// TIA Portal V17 export
// export: Created 2026-04-13T11:12:44.2249496Z, ExportSetting WithDefaults, DisplayName Totally Integrated Automation Portal, DisplayVersion V17 Update 4, DisplayName TIA Portal Openness, DisplayVersion V17 Update 4, DisplayName TIA Portal Version Control Interface, DisplayVersion V17, DisplayName SINAMICS Startdrive Advanced, DisplayVersion V17, DisplayName SINAMICS Startdrive G130, G150, S120, S150, SINAMICS MV, S210, DisplayVersion V17, DisplayName SINAMICS Startdrive G110M, G120, G120C, G120D, G120P, G115D, DisplayVersion V17, DisplayName STEP 7 Professional, DisplayVersion V17 Update 4, DisplayName STEP 7 Safety, DisplayVersion V17, DisplayName WinCC Professional, DisplayVersion V17 Update 4
FUNCTION_BLOCK "16-普通脉冲"   // FB53, SCL
{ S7_Optimized_Access := 'TRUE' }
VERSION : 0.1
// stored: AutoNumber true, IsIECCheckEnabled false, IsRetainMemResEnabled false, MemoryReserve 100, SetENOAutomatically false, UDAEnableTagReadback false
   VAR_INPUT
      模式设定 : Real;
      QD : Bool;
      On_Time : Real;
      Stop_Time : Real;
      Num : Int;
   END_VAR
   VAR_OUTPUT
      Output_1 : Bool;
      Output_2 : Bool;
      Output_3 : Bool;
      Output_4 : Bool;
      Output_5 : Bool;
      Output_6 : Bool;
      Output_7 : Bool;
      Output_8 : Bool;
      Num_now : Int;
   END_VAR
   VAR
      Stoptime : Time;
      WorkTime : Time;
      TON_ON : Array[1..10] of TON_TIME;
      TON_OFF : Array[1..10] of TON_TIME;
   END_VAR
BEGIN

   IF #模式设定 = 1.0  OR #模式设定 = 2.0  THEN
       #Stoptime := DINT_TO_TIME(REAL_TO_DINT(#Stop_Time * 1000.0));
       //#WorkTime := DINT_TO_TIME(REAL_TO_DINT(#On_Time * 1000));
        #WorkTime := REAL_TO_DINT(#On_Time);

       IF NOT #QD THEN
           #Num_now := 0;
       ELSE

           IF #Num <= 12 THEN
               #Num_now := #Num;
           ELSE
               #Num_now := 12;
           END_IF;

       END_IF;



       CASE #Num_now OF
           1:
               #TON_ON[1](IN := #QD AND NOT #TON_OFF[1].Q,
                          PT := #WorkTime);
               #TON_OFF[1](IN := #QD AND #TON_ON[1].Q,
                           PT := #Stoptime);


               #Output_1 := #QD AND NOT #TON_ON[1].Q;


           2:  // Statement section case 1
               #TON_ON[1](IN := #QD AND NOT #TON_OFF[2].Q,
                          PT := #WorkTime);
               #TON_OFF[1](IN := #QD AND #TON_ON[1].Q,
                           PT := #Stoptime);
               #TON_ON[2](IN := #QD AND #TON_ON[1].Q AND #TON_OFF[1].Q,
                          PT := #WorkTime);
               #TON_OFF[2](IN := #QD AND #TON_ON[1].Q AND #TON_OFF[1].Q AND #TON_ON[2].Q,
                           PT := #Stoptime);

               #Output_1 := #QD AND NOT #TON_ON[1].Q;
               #Output_2 := #QD AND #TON_ON[1].Q AND #TON_OFF[1].Q AND NOT #TON_ON[2].Q;

           3:  // Statement section case 2 to 4
               #TON_ON[1](IN := #QD AND NOT #TON_OFF[3].Q,
                          PT := #WorkTime);
               #TON_OFF[1](IN := #QD AND #TON_ON[1].Q,
                           PT := #Stoptime);
               #TON_ON[2](IN := #QD AND #TON_ON[1].Q AND #TON_OFF[1].Q,
                          PT := #WorkTime);
               #TON_OFF[2](IN := #QD AND #TON_ON[1].Q AND #TON_OFF[1].Q AND #TON_ON[2].Q,
                           PT := #Stoptime);
               #TON_ON[3](IN := #QD AND #TON_ON[1].Q AND #TON_OFF[1].Q AND #TON_ON[2].Q AND #TON_OFF[2].Q,
                          PT := #WorkTime);
               #TON_OFF[3](IN := #QD AND #TON_ON[1].Q AND #TON_OFF[1].Q AND #TON_ON[2].Q AND #TON_OFF[2].Q AND #TON_ON[3].Q,
                           PT := #Stoptime);
               #Output_1 := #QD AND NOT #TON_ON[1].Q;
               #Output_2 := #QD AND #TON_ON[1].Q AND #TON_OFF[1].Q AND NOT #TON_ON[2].Q;
               #Output_3 := #QD AND #TON_ON[1].Q AND #TON_OFF[1].Q AND #TON_ON[2].Q AND #TON_OFF[2].Q AND NOT #TON_ON[3].Q;
           4:  // Statement section case 2 to 4
               #TON_ON[1](IN := #QD AND NOT #TON_OFF[4].Q,
                          PT := #WorkTime);
               #TON_OFF[1](IN := #QD AND #TON_ON[1].Q,
                           PT := #Stoptime);
               #TON_ON[2](IN := #QD AND #TON_ON[1].Q AND #TON_OFF[1].Q,
                          PT := #WorkTime);
               #TON_OFF[2](IN := #QD AND #TON_ON[1].Q AND #TON_OFF[1].Q AND #TON_ON[2].Q,
                           PT := #Stoptime);
               #TON_ON[3](IN := #QD AND #TON_ON[1].Q AND #TON_OFF[1].Q AND #TON_ON[2].Q AND #TON_OFF[2].Q,
                          PT := #WorkTime);
               #TON_OFF[3](IN := #QD AND #TON_ON[1].Q AND #TON_OFF[1].Q AND #TON_ON[2].Q AND #TON_OFF[2].Q AND #TON_ON[3].Q,
                           PT := #Stoptime);

               #TON_ON[4](IN := #QD AND #TON_ON[1].Q AND #TON_OFF[1].Q AND #TON_ON[2].Q AND #TON_OFF[2].Q AND #TON_ON[3].Q AND #TON_OFF[3].Q,
                          PT := #WorkTime);
               #TON_OFF[4](IN := #QD AND #TON_ON[1].Q AND #TON_OFF[1].Q AND #TON_ON[2].Q AND #TON_OFF[2].Q AND #TON_ON[3].Q AND #TON_OFF[3].Q AND #TON_ON[4].Q,
                           PT := #Stoptime);


               #Output_1 := #QD AND NOT #TON_ON[1].Q;
               #Output_2 := #QD AND #TON_ON[1].Q AND #TON_OFF[1].Q AND NOT #TON_ON[2].Q;
               #Output_3 := #QD AND #TON_ON[1].Q AND #TON_OFF[1].Q AND #TON_ON[2].Q AND #TON_OFF[2].Q AND NOT #TON_ON[3].Q;
               #Output_4 := #QD AND #TON_ON[1].Q AND #TON_OFF[1].Q AND #TON_ON[2].Q AND #TON_OFF[2].Q AND #TON_ON[3].Q AND #TON_OFF[3].Q AND NOT #TON_ON[4].Q;

           5:  // Statement section case 2 to 4
               #TON_ON[1](IN := #QD AND NOT #TON_OFF[5].Q,
                          PT := #WorkTime);
               #TON_OFF[1](IN := #QD AND #TON_ON[1].Q,
                           PT := #Stoptime);
               #TON_ON[2](IN := #QD AND #TON_ON[1].Q AND #TON_OFF[1].Q,
                          PT := #WorkTime);
               #TON_OFF[2](IN := #QD AND #TON_ON[1].Q AND #TON_OFF[1].Q AND #TON_ON[2].Q,
                           PT := #Stoptime);
               #TON_ON[3](IN := #QD AND #TON_ON[1].Q AND #TON_OFF[1].Q AND #TON_ON[2].Q AND #TON_OFF[2].Q,
                          PT := #WorkTime);
               #TON_OFF[3](IN := #QD AND #TON_ON[1].Q AND #TON_OFF[1].Q AND #TON_ON[2].Q AND #TON_OFF[2].Q AND #TON_ON[3].Q,
                           PT := #Stoptime);

               #TON_ON[4](IN := #QD AND #TON_ON[1].Q AND #TON_OFF[1].Q AND #TON_ON[2].Q AND #TON_OFF[2].Q AND #TON_ON[3].Q AND #TON_OFF[3].Q,
                          PT := #WorkTime);
               #TON_OFF[4](IN := #QD AND #TON_ON[1].Q AND #TON_OFF[1].Q AND #TON_ON[2].Q AND #TON_OFF[2].Q AND #TON_ON[3].Q AND #TON_OFF[3].Q AND #TON_ON[4].Q,
                           PT := #Stoptime);

               #TON_ON[5](IN := #QD AND #TON_ON[1].Q AND #TON_OFF[1].Q AND #TON_ON[2].Q AND #TON_OFF[2].Q AND #TON_ON[3].Q AND #TON_OFF[3].Q AND #TON_ON[4].Q AND #TON_OFF[4].Q,
                          PT := #WorkTime);
               #TON_OFF[5](IN := #QD AND #TON_ON[1].Q AND #TON_OFF[1].Q AND #TON_ON[2].Q AND #TON_OFF[2].Q AND #TON_ON[3].Q AND #TON_OFF[3].Q AND #TON_ON[4].Q AND #TON_OFF[4].Q AND #TON_ON[5].Q,
                           PT := #Stoptime);


               #Output_1 := #QD AND NOT #TON_ON[1].Q;
               #Output_2 := #QD AND #TON_ON[1].Q AND #TON_OFF[1].Q AND NOT #TON_ON[2].Q;
               #Output_3 := #QD AND #TON_ON[1].Q AND #TON_OFF[1].Q AND #TON_ON[2].Q AND #TON_OFF[2].Q AND NOT #TON_ON[3].Q;
               #Output_4 := #QD AND #TON_ON[1].Q AND #TON_OFF[1].Q AND #TON_ON[2].Q AND #TON_OFF[2].Q AND #TON_ON[3].Q AND #TON_OFF[3].Q AND NOT #TON_ON[4].Q;
               #Output_5 := #QD AND #TON_ON[1].Q AND #TON_OFF[1].Q AND #TON_ON[2].Q AND #TON_OFF[2].Q AND #TON_ON[3].Q AND #TON_OFF[3].Q AND #TON_ON[4].Q AND #TON_OFF[4].Q AND NOT #TON_ON[5].Q;

           6:  // Statement section case 2 to 4
               #TON_ON[1](IN := #QD AND NOT #TON_OFF[6].Q,
                          PT := #WorkTime);
               #TON_OFF[1](IN := #QD AND #TON_ON[1].Q,
                           PT := #Stoptime);
               #TON_ON[2](IN := #QD AND #TON_ON[1].Q AND #TON_OFF[1].Q,
                          PT := #WorkTime);
               #TON_OFF[2](IN := #QD AND #TON_ON[1].Q AND #TON_OFF[1].Q AND #TON_ON[2].Q,
                           PT := #Stoptime);
               #TON_ON[3](IN := #QD AND #TON_ON[1].Q AND #TON_OFF[1].Q AND #TON_ON[2].Q AND #TON_OFF[2].Q,
                          PT := #WorkTime);
               #TON_OFF[3](IN := #QD AND #TON_ON[1].Q AND #TON_OFF[1].Q AND #TON_ON[2].Q AND #TON_OFF[2].Q AND #TON_ON[3].Q,
                           PT := #Stoptime);

               #TON_ON[4](IN := #QD AND #TON_ON[1].Q AND #TON_OFF[1].Q AND #TON_ON[2].Q AND #TON_OFF[2].Q AND #TON_ON[3].Q AND #TON_OFF[3].Q,
                          PT := #WorkTime);
               #TON_OFF[4](IN := #QD AND #TON_ON[1].Q AND #TON_OFF[1].Q AND #TON_ON[2].Q AND #TON_OFF[2].Q AND #TON_ON[3].Q AND #TON_OFF[3].Q AND #TON_ON[4].Q,
                           PT := #Stoptime);

               #TON_ON[5](IN := #QD AND #TON_ON[1].Q AND #TON_OFF[1].Q AND #TON_ON[2].Q AND #TON_OFF[2].Q AND #TON_ON[3].Q AND #TON_OFF[3].Q AND #TON_ON[4].Q AND #TON_OFF[4].Q,
                          PT := #WorkTime);
               #TON_OFF[5](IN := #QD AND #TON_ON[1].Q AND #TON_OFF[1].Q AND #TON_ON[2].Q AND #TON_OFF[2].Q AND #TON_ON[3].Q AND #TON_OFF[3].Q AND #TON_ON[4].Q AND #TON_OFF[4].Q AND #TON_ON[5].Q,
                           PT := #Stoptime);

               #TON_ON[6](IN := #QD AND #TON_ON[1].Q AND #TON_OFF[1].Q AND #TON_ON[2].Q AND #TON_OFF[2].Q AND #TON_ON[3].Q AND #TON_OFF[3].Q AND #TON_ON[4].Q AND #TON_OFF[4].Q AND #TON_ON[5].Q AND #TON_OFF[5].Q,
                          PT := #WorkTime);
               #TON_OFF[6](IN := #QD AND #TON_ON[1].Q AND #TON_OFF[1].Q AND #TON_ON[2].Q AND #TON_OFF[2].Q AND #TON_ON[3].Q AND #TON_OFF[3].Q AND #TON_ON[4].Q AND #TON_OFF[4].Q AND #TON_ON[5].Q AND #TON_OFF[5].Q AND #TON_ON[6].Q,
                           PT := #Stoptime);


               #Output_1 := #QD AND NOT #TON_ON[1].Q;
               #Output_2 := #QD AND #TON_ON[1].Q AND #TON_OFF[1].Q AND NOT #TON_ON[2].Q;
               #Output_3 := #QD AND #TON_ON[1].Q AND #TON_OFF[1].Q AND #TON_ON[2].Q AND #TON_OFF[2].Q AND NOT #TON_ON[3].Q;
               #Output_4 := #QD AND #TON_ON[1].Q AND #TON_OFF[1].Q AND #TON_ON[2].Q AND #TON_OFF[2].Q AND #TON_ON[3].Q AND #TON_OFF[3].Q AND NOT #TON_ON[4].Q;
               #Output_5 := #QD AND #TON_ON[1].Q AND #TON_OFF[1].Q AND #TON_ON[2].Q AND #TON_OFF[2].Q AND #TON_ON[3].Q AND #TON_OFF[3].Q AND #TON_ON[4].Q AND #TON_OFF[4].Q AND NOT #TON_ON[5].Q;
               #Output_6 := #QD AND #TON_ON[1].Q AND #TON_OFF[1].Q AND #TON_ON[2].Q AND #TON_OFF[2].Q AND #TON_ON[3].Q AND #TON_OFF[3].Q AND #TON_ON[4].Q AND #TON_OFF[4].Q AND #TON_ON[5].Q AND #TON_OFF[5].Q AND NOT #TON_ON[6].Q;

           7:  // Statement section case 2 to 4
               #TON_ON[1](IN := #QD AND NOT #TON_OFF[7].Q,
                          PT := #WorkTime);
               #TON_OFF[1](IN := #QD AND #TON_ON[1].Q,
                           PT := #Stoptime);
               #TON_ON[2](IN := #QD AND #TON_ON[1].Q AND #TON_OFF[1].Q,
                          PT := #WorkTime);
               #TON_OFF[2](IN := #QD AND #TON_ON[1].Q AND #TON_OFF[1].Q AND #TON_ON[2].Q,
                           PT := #Stoptime);
               #TON_ON[3](IN := #QD AND #TON_ON[1].Q AND #TON_OFF[1].Q AND #TON_ON[2].Q AND #TON_OFF[2].Q,
                          PT := #WorkTime);
               #TON_OFF[3](IN := #QD AND #TON_ON[1].Q AND #TON_OFF[1].Q AND #TON_ON[2].Q AND #TON_OFF[2].Q AND #TON_ON[3].Q,
                           PT := #Stoptime);

               #TON_ON[4](IN := #QD AND #TON_ON[1].Q AND #TON_OFF[1].Q AND #TON_ON[2].Q AND #TON_OFF[2].Q AND #TON_ON[3].Q AND #TON_OFF[3].Q,
                          PT := #WorkTime);
               #TON_OFF[4](IN := #QD AND #TON_ON[1].Q AND #TON_OFF[1].Q AND #TON_ON[2].Q AND #TON_OFF[2].Q AND #TON_ON[3].Q AND #TON_OFF[3].Q AND #TON_ON[4].Q,
                           PT := #Stoptime);

               #TON_ON[5](IN := #QD AND #TON_ON[1].Q AND #TON_OFF[1].Q AND #TON_ON[2].Q AND #TON_OFF[2].Q AND #TON_ON[3].Q AND #TON_OFF[3].Q AND #TON_ON[4].Q AND #TON_OFF[4].Q,
                          PT := #WorkTime);
               #TON_OFF[5](IN := #QD AND #TON_ON[1].Q AND #TON_OFF[1].Q AND #TON_ON[2].Q AND #TON_OFF[2].Q AND #TON_ON[3].Q AND #TON_OFF[3].Q AND #TON_ON[4].Q AND #TON_OFF[4].Q AND #TON_ON[5].Q,
                           PT := #Stoptime);

               #TON_ON[6](IN := #QD AND #TON_ON[1].Q AND #TON_OFF[1].Q AND #TON_ON[2].Q AND #TON_OFF[2].Q AND #TON_ON[3].Q AND #TON_OFF[3].Q AND #TON_ON[4].Q AND #TON_OFF[4].Q AND #TON_ON[5].Q AND #TON_OFF[5].Q,
                          PT := #WorkTime);
               #TON_OFF[6](IN := #QD AND #TON_ON[1].Q AND #TON_OFF[1].Q AND #TON_ON[2].Q AND #TON_OFF[2].Q AND #TON_ON[3].Q AND #TON_OFF[3].Q AND #TON_ON[4].Q AND #TON_OFF[4].Q AND #TON_ON[5].Q AND #TON_OFF[5].Q AND #TON_ON[6].Q,
                           PT := #Stoptime);

               #TON_ON[7](IN := #QD AND #TON_ON[1].Q AND #TON_OFF[1].Q AND #TON_ON[2].Q AND #TON_OFF[2].Q AND #TON_ON[3].Q AND #TON_OFF[3].Q AND #TON_ON[4].Q AND #TON_OFF[5].Q AND #TON_ON[5].Q AND #TON_OFF[6].Q AND #TON_ON[6].Q AND #TON_OFF[6].Q,
                          PT := #WorkTime);
               #TON_OFF[7](IN := #QD AND #TON_ON[1].Q AND #TON_OFF[1].Q AND #TON_ON[2].Q AND #TON_OFF[2].Q AND #TON_ON[3].Q AND #TON_OFF[3].Q AND #TON_ON[4].Q AND #TON_OFF[5].Q AND #TON_ON[5].Q AND #TON_OFF[6].Q AND #TON_ON[6].Q AND #TON_OFF[6].Q AND #TON_ON[7].Q,
                           PT := #Stoptime);



               #Output_1 := #QD AND NOT #TON_ON[1].Q;
               #Output_2 := #QD AND #TON_ON[1].Q AND #TON_OFF[1].Q AND NOT #TON_ON[2].Q;
               #Output_3 := #QD AND #TON_ON[1].Q AND #TON_OFF[1].Q AND #TON_ON[2].Q AND #TON_OFF[2].Q AND NOT #TON_ON[3].Q;
               #Output_4 := #QD AND #TON_ON[1].Q AND #TON_OFF[1].Q AND #TON_ON[2].Q AND #TON_OFF[2].Q AND #TON_ON[3].Q AND #TON_OFF[3].Q AND NOT #TON_ON[4].Q;
               #Output_5 := #QD AND #TON_ON[1].Q AND #TON_OFF[1].Q AND #TON_ON[2].Q AND #TON_OFF[2].Q AND #TON_ON[3].Q AND #TON_OFF[3].Q AND #TON_ON[4].Q AND #TON_OFF[4].Q AND NOT #TON_ON[5].Q;
               #Output_6 := #QD AND #TON_ON[1].Q AND #TON_OFF[1].Q AND #TON_ON[2].Q AND #TON_OFF[2].Q AND #TON_ON[3].Q AND #TON_OFF[3].Q AND #TON_ON[4].Q AND #TON_OFF[4].Q AND #TON_ON[5].Q AND #TON_OFF[5].Q AND NOT #TON_ON[6].Q;
               #Output_7 := #QD AND #TON_ON[1].Q AND #TON_OFF[1].Q AND #TON_ON[2].Q AND #TON_OFF[2].Q AND #TON_ON[3].Q AND #TON_OFF[3].Q AND #TON_ON[4].Q AND #TON_OFF[4].Q AND #TON_ON[5].Q AND #TON_OFF[5].Q AND #TON_ON[6].Q AND #TON_OFF[6].Q AND NOT #TON_ON[7].Q;

           8:  // Statement section case 2 to 4
               #TON_ON[1](IN := #QD AND NOT #TON_OFF[8].Q,
                          PT := #WorkTime);
               #TON_OFF[1](IN := #QD AND #TON_ON[1].Q,
                           PT := #Stoptime);
               #TON_ON[2](IN := #QD AND #TON_ON[1].Q AND #TON_OFF[1].Q,
                          PT := #WorkTime);
               #TON_OFF[2](IN := #QD AND #TON_ON[1].Q AND #TON_OFF[1].Q AND #TON_ON[2].Q,
                           PT := #Stoptime);
               #TON_ON[3](IN := #QD AND #TON_ON[1].Q AND #TON_OFF[1].Q AND #TON_ON[2].Q AND #TON_OFF[2].Q,
                          PT := #WorkTime);
               #TON_OFF[3](IN := #QD AND #TON_ON[1].Q AND #TON_OFF[1].Q AND #TON_ON[2].Q AND #TON_OFF[2].Q AND #TON_ON[3].Q,
                           PT := #Stoptime);

               #TON_ON[4](IN := #QD AND #TON_ON[1].Q AND #TON_OFF[1].Q AND #TON_ON[2].Q AND #TON_OFF[2].Q AND #TON_ON[3].Q AND #TON_OFF[3].Q,
                          PT := #WorkTime);
               #TON_OFF[4](IN := #QD AND #TON_ON[1].Q AND #TON_OFF[1].Q AND #TON_ON[2].Q AND #TON_OFF[2].Q AND #TON_ON[3].Q AND #TON_OFF[3].Q AND #TON_ON[4].Q,
                           PT := #Stoptime);

               #TON_ON[5](IN := #QD AND #TON_ON[1].Q AND #TON_OFF[1].Q AND #TON_ON[2].Q AND #TON_OFF[2].Q AND #TON_ON[3].Q AND #TON_OFF[3].Q AND #TON_ON[4].Q AND #TON_OFF[4].Q,
                          PT := #WorkTime);
               #TON_OFF[5](IN := #QD AND #TON_ON[1].Q AND #TON_OFF[1].Q AND #TON_ON[2].Q AND #TON_OFF[2].Q AND #TON_ON[3].Q AND #TON_OFF[3].Q AND #TON_ON[4].Q AND #TON_OFF[4].Q AND #TON_ON[5].Q,
                           PT := #Stoptime);

               #TON_ON[6](IN := #QD AND #TON_ON[1].Q AND #TON_OFF[1].Q AND #TON_ON[2].Q AND #TON_OFF[2].Q AND #TON_ON[3].Q AND #TON_OFF[3].Q AND #TON_ON[4].Q AND #TON_OFF[4].Q AND #TON_ON[5].Q AND #TON_OFF[5].Q,
                          PT := #WorkTime);
               #TON_OFF[6](IN := #QD AND #TON_ON[1].Q AND #TON_OFF[1].Q AND #TON_ON[2].Q AND #TON_OFF[2].Q AND #TON_ON[3].Q AND #TON_OFF[3].Q AND #TON_ON[4].Q AND #TON_OFF[4].Q AND #TON_ON[5].Q AND #TON_OFF[5].Q AND #TON_ON[6].Q,
                           PT := #Stoptime);

               #TON_ON[7](IN := #QD AND #TON_ON[1].Q AND #TON_OFF[1].Q AND #TON_ON[2].Q AND #TON_OFF[2].Q AND #TON_ON[3].Q AND #TON_OFF[3].Q AND #TON_ON[4].Q AND #TON_OFF[4].Q AND #TON_ON[5].Q AND #TON_OFF[5].Q AND #TON_ON[6].Q AND #TON_OFF[6].Q,
                          PT := #WorkTime);
               #TON_OFF[7](IN := #QD AND #TON_ON[1].Q AND #TON_OFF[1].Q AND #TON_ON[2].Q AND #TON_OFF[2].Q AND #TON_ON[3].Q AND #TON_OFF[3].Q AND #TON_ON[4].Q AND #TON_OFF[4].Q AND #TON_ON[5].Q AND #TON_OFF[5].Q AND #TON_ON[6].Q AND #TON_OFF[6].Q AND #TON_ON[7].Q,
                           PT := #Stoptime);
               #TON_ON[8](IN := #QD AND #TON_ON[1].Q AND #TON_OFF[1].Q AND #TON_ON[2].Q AND #TON_OFF[2].Q AND #TON_ON[3].Q AND #TON_OFF[3].Q AND #TON_ON[4].Q AND #TON_OFF[4].Q AND #TON_ON[5].Q AND #TON_OFF[5].Q AND #TON_ON[6].Q AND #TON_OFF[6].Q AND #TON_ON[7].Q AND #TON_OFF[7].Q,
                          PT := #WorkTime);
               #TON_OFF[8](IN := #QD AND #TON_ON[1].Q AND #TON_OFF[1].Q AND #TON_ON[2].Q AND #TON_OFF[2].Q AND #TON_ON[3].Q AND #TON_OFF[3].Q AND #TON_ON[4].Q AND #TON_OFF[4].Q AND #TON_ON[5].Q AND #TON_OFF[5].Q AND #TON_ON[6].Q AND #TON_OFF[6].Q AND #TON_ON[7].Q AND #TON_OFF[7].Q AND #TON_ON[8].Q,
                           PT := #Stoptime);


               #Output_1 := #QD AND NOT #TON_ON[1].Q;
               #Output_2 := #QD AND #TON_ON[1].Q AND #TON_OFF[1].Q AND NOT #TON_ON[2].Q;
               #Output_3 := #QD AND #TON_ON[1].Q AND #TON_OFF[1].Q AND #TON_ON[2].Q AND #TON_OFF[2].Q AND NOT #TON_ON[3].Q;
               #Output_4 := #QD AND #TON_ON[1].Q AND #TON_OFF[1].Q AND #TON_ON[2].Q AND #TON_OFF[2].Q AND #TON_ON[3].Q AND #TON_OFF[3].Q AND NOT #TON_ON[4].Q;
               #Output_5 := #QD AND #TON_ON[1].Q AND #TON_OFF[1].Q AND #TON_ON[2].Q AND #TON_OFF[2].Q AND #TON_ON[3].Q AND #TON_OFF[3].Q AND #TON_ON[4].Q AND #TON_OFF[4].Q AND NOT #TON_ON[5].Q;
               #Output_6 := #QD AND #TON_ON[1].Q AND #TON_OFF[1].Q AND #TON_ON[2].Q AND #TON_OFF[2].Q AND #TON_ON[3].Q AND #TON_OFF[3].Q AND #TON_ON[4].Q AND #TON_OFF[4].Q AND #TON_ON[5].Q AND #TON_OFF[5].Q AND NOT #TON_ON[6].Q;
               #Output_7 := #QD AND #TON_ON[1].Q AND #TON_OFF[1].Q AND #TON_ON[2].Q AND #TON_OFF[2].Q AND #TON_ON[3].Q AND #TON_OFF[3].Q AND #TON_ON[4].Q AND #TON_OFF[4].Q AND #TON_ON[5].Q AND #TON_OFF[5].Q AND #TON_ON[6].Q AND #TON_OFF[6].Q AND NOT #TON_ON[7].Q;
               #Output_8 := #QD AND #TON_ON[1].Q AND #TON_OFF[1].Q AND #TON_ON[2].Q AND #TON_OFF[2].Q AND #TON_ON[3].Q AND #TON_OFF[3].Q AND #TON_ON[4].Q AND #TON_OFF[4].Q AND #TON_ON[5].Q AND #TON_OFF[5].Q AND #TON_ON[6].Q AND #TON_OFF[6].Q AND #TON_ON[7].Q AND #TON_OFF[7].Q AND NOT #TON_ON[8].Q;

           ELSE  // Statement section ELSE
               ;
       END_CASE;
   END_IF;


   IF NOT #QD THEN

       #Output_1 := 0;
       #Output_2 := 0;
       #Output_3 := 0;
       #Output_4 := 0;
       #Output_5 := 0;
       #Output_6 := 0;
       #Output_7 := 0;
       #Output_8 := 0;
   END_IF;
END_FUNCTION_BLOCK
